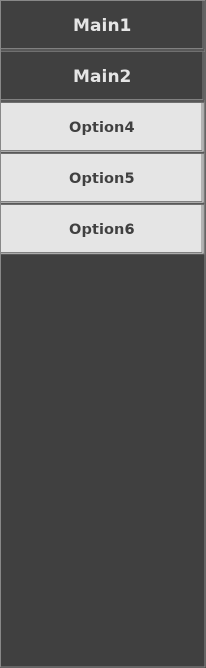
VISUALIZATION PH_Menu  // 206x668
VAR_IN_OUT
	bMain1									: BOOL;
	bMain2									: BOOL;
	iFrameNumber							: INT;
	udiFOntColor1 							: UDINT;
	udiFontColor2							: UDINT;
END_VAR
    Group (0,0 206x254), invisible if: NOT GVL_HMI.bMenu
        Group (0,51 206x152), invisible if: NOT bMain1
            Button (0,0 204x50), "File Dialog"
                OnMouseDown: execute { GVL_HMI.iFrameNumber:=5; GVL_HMI.bMenu:=FALSE; }
            Button (0,102 204x50), "Trends"
                OnMouseDown: execute { GVL_HMI.iFrameNumber:=7; GVL_HMI.bMenu:=FALSE; }
            Button (0,51 204x50), "Table"
                OnMouseDown: execute { GVL_HMI.iFrameNumber:=6; GVL_HMI.bMenu:=FALSE; }
        Group (0,102 206x152), invisible if: NOT bMain2
            Button (0,102 204x50), "Option6"
                OnMouseDown: execute { GVL_HMI.iFrameNumber:=10; GVL_HMI.bMenu:=FALSE; }
            Button (0,51 204x50), "Option5"
                OnMouseDown: execute { GVL_HMI.iFrameNumber:=9; GVL_HMI.bMenu:=FALSE; }
            Button (0,0 204x50), "Option4"
                OnMouseDown: execute { GVL_HMI.iFrameNumber:=8; GVL_HMI.bMenu:=FALSE; }
        Button (0,51 205x50), "Main2", colour toggle: bMain2
            p2738717112: BOOL_TO_INT(bMain1)*153
            p55702900: udiFontColor2
            OnMouseDown: execute { GVL_Hmi.bMain1:=FALSE; GVL_HMI.bMain2:=TRUE; }
        Button (0,0 205x50), "Main1", colour toggle: bMain1
            p55702900: udiFOntColor1
            OnMouseDown: execute { GVL_HMI.bMain2:=FALSE; GVL_HMI.bMain1:=TRUE; }
END_VISUALIZATION

(* stored: Version 1.1.0.1, ProductVersion 3.1.4024.3
   Visu PH_Menu: Id {12f38f62-f595-4557-94ce-440c2bf1266d} *)
